{attribute 'GeneratedUsingTerminal: EL2642-0000-0016'}
{attribute addProperty BoxType "EL2642-0000-0016"}
{attribute addProperty Id "Outputs_Group_1AT %Q*Outputs_Group_78994C084"}
{attribute addProperty CRC "1507377180"}
{attribute addProperty Size "4"}
TYPE DO_Group_1_Outputs_59D8C01C :
STRUCT
	{attribute addProperty Name "Outputs_Group_1"}
	Outputs_Group_1 AT %Q* : Outputs_Group_78994C08;
END_STRUCT
END_TYPE

(* stored: Version 1.2.0.0, ProductVersion 3.1.4024.9
   DUT DO_Group_1_Outputs_59D8C01C: Id {ff1526c3-601e-43f2-b00f-c2281db5823a} *)
